Universal Robots URScript: force01.script

# force
# movej
# waypoint 1
# waypoint 2

def unnamed():
  global _hidden_verificationVariable=0
  step_count_f5b51f0c_4365_410e_844e_85abb40d34c3 = 0.0
  thread Step_Counter_Thread_6336083a_980d_4b96_bd1e_426122f1dec4():
    while (True):
      step_count_f5b51f0c_4365_410e_844e_85abb40d34c3 = step_count_f5b51f0c_4365_410e_844e_85abb40d34c3 + 1.0
      sync()
    end
  end
  run Step_Counter_Thread_6336083a_980d_4b96_bd1e_426122f1dec4()
  set_gravity([0.0, 0.0, 9.82])
  set_safety_mode_transition_hardness(1)
  set_target_payload(1.000000, [0.000000, 0.000000, 0.000000], [0.001539, 0.001539, 0.001539, 0.000000, 0.000000, 0.000000])
  set_tcp(p[0.0,0.0,0.0,0.0,0.0,0.0])
  set_tool_communication(False, 115200, 0, 1, 1.5, 3.5)
  set_tool_output_mode(0)
  set_tool_digital_output_mode(0, 1)
  set_tool_digital_output_mode(1, 1)
  set_tool_voltage(0)
  set_standard_analog_input_domain(0, 1)
  set_standard_analog_input_domain(1, 1)
  set_tool_analog_input_domain(0, 1)
  set_tool_analog_input_domain(1, 1)
  set_analog_outputdomain(0, 0)
  set_analog_outputdomain(1, 0)
  set_input_actions_to_default()
  global i_var_1=10
  global Waypoint_1_p=p[.233984917120, -.298943670708, .323871260948, -.371542170508, 3.097153373370, .043298329506]
  global Waypoint_1_q=[-0.5633569741221507, -1.8233190611528212, -1.185235347866847, -1.7043312223477276, 1.6061707300222556, 0.7686467091801763]
  global Waypoint_2_p=p[.303736482787, -.255560701535, .323871260935, -.371542170508, 3.097153373367, .043298329511]
  global Waypoint_2_q=[-0.37156168762027875, -1.9023567130266272, -1.0826669175192727, -1.7211070365931178, 1.6056164978469303, 0.9605597500982175]
  while (True):
    $ 1 "Robot Program"
    $ 2 "Force"
    sleep(0.02)
    zero_ftsensor()
    force_mode(p[0.0,0.0,0.0,0.0,0.0,0.0], [0, 0, 1, 0, 0, 0], [0.0, 0.0, 0.0, 0.0, 0.0, 0.0], 2, [0.1, 0.1, 0.15, 0.3490658503988659, 0.3490658503988659, 0.3490658503988659])
    $ 3 "MoveJ" "noBreak"
    $ 4 "Waypoint_1" "noBreak"
    movej(get_inverse_kin(Waypoint_1_p, qnear=Waypoint_1_q), a=1.3962634015954636, v=1.0471975511965976)
    $ 5 "Waypoint_2" "noBreak"
    movej(get_inverse_kin(Waypoint_2_p, qnear=Waypoint_2_q), a=1.3962634015954636, v=1.0471975511965976)
    end_force_mode()
    stopl(5.0)
  end
end
